// TIA Portal V17 export
// export: Created 2025-07-17T00:36:38.1695794Z, ExportSetting WithDefaults, DisplayName Totally Integrated Automation Portal, DisplayVersion V17, DisplayName TIA Portal Openness, DisplayVersion V17, DisplayName TIA Portal Version Control Interface, DisplayVersion V17, DisplayName STEP 7 Professional, DisplayVersion V17, DisplayName STEP 7 Safety, DisplayVersion V17, DisplayName WinCC Advanced / Unified PC, DisplayVersion V17
FUNCTION_BLOCK "pump_flow_set"   // FB2, LAD
{ S7_Optimized_Access := 'TRUE' }
VERSION : 0.1
// stored: AutoNumber true, IsIECCheckEnabled false, IsRetainMemResEnabled false, MemoryReserve 100, SetENOAutomatically false, UDAEnableTagReadback false
   VAR_INPUT
      local_remote : Bool;
      local_flow_set : Real;
      remote_flow_set : Real;
   END_VAR
   VAR_OUTPUT
      flow_set_output : Real;
   END_VAR
   VAR_TEMP
      control_flow : Real;
      flow_temp_real : Real;
   END_VAR
BEGIN

REGION Network 1
   // 远程/在地切换
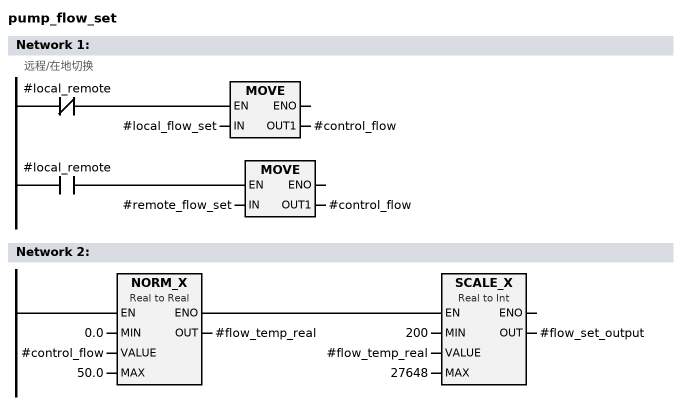
   RUNG wire#powerrail
      I_Contact( #local_remote )
      Move(in := #local_flow_set, out1 => #control_flow)
   END_RUNG
   RUNG wire#powerrail
      Contact( #local_remote )
      Move(in := #remote_flow_set, out1 => #control_flow)
   END_RUNG
   // the same network as SCL:
   IF NOT #local_remote THEN #control_flow := #local_flow_set; END_IF;
   IF #local_remote THEN #control_flow := #remote_flow_set; END_IF;
END_REGION

REGION Network 2
   RUNG wire#powerrail
      { S7_Templates := "[SrcType := Real, DestType := Real]" } Normalize(min := 0.0, value := #control_flow, max := 50.0, out => #flow_temp_real)
      { S7_Templates := "[SrcType := Real, DestType := Int]" } Scale(min := 200, value := #flow_temp_real, max := 27648, out => #flow_set_output)
   END_RUNG
   // the same network as SCL:
   #flow_temp_real := NORM_X(MIN := 0.0, VALUE := #control_flow, MAX := 50.0);
   #flow_set_output := SCALE_X(MIN := 200, VALUE := #flow_temp_real, MAX := 27648);
END_REGION
END_FUNCTION_BLOCK
